// TIA Portal V17 export
// export: Created 2023-10-17T06:55:21.0718728Z, ExportSetting WithDefaults, DisplayName Totally Integrated Automation Portal, DisplayVersion V17, DisplayName TIA Portal Openness, DisplayVersion V17, DisplayName TIA Portal Version Control Interface, DisplayVersion V17, DisplayName STEP 7 Professional, DisplayVersion V17, DisplayName STEP 7 Safety, DisplayVersion V17, DisplayName WinCC Advanced, DisplayVersion V17
DATA_BLOCK "Recipe_Parameter"   // DB2
{ S7_Optimized_Access := 'FALSE' }
VERSION : 0.1
// stored: AutoNumber true, DBAccessibleFromOPCUA true, DBAccessibleFromWebserver true, IsOnlyStoredInLoadMemory false, IsWriteProtectedInAS false
   VAR
      SelectedFlavor : Int;
      Milk_Volume : Real;
      Flavor_Volume : Real;
      Mixing_Time : Time;
      Pasteurising_Time : Time;
   END_VAR
BEGIN
END_DATA_BLOCK
